  rq_init_comm_if_connected(9, "1")
  rq_init_comm_if_connected(2, "2")
  rq_init_comm_if_connected(3, "3")
  rq_init_comm_if_connected(4, "4")
  rq_print_connected_grippers()
  rq_gripper_communication_thread = run rq_gripper_communication()
  set_closed_norm(100.0, 1)
  set_open_norm(0.0, 1)
  set_closed_mm(0.0, 1)
  set_open_mm(50.0, 1)
  set_closed_norm(100.0, 2)
  set_open_norm(0.0, 2)
  set_closed_mm(0.0, 2)
  set_open_mm(50.0, 2)
  set_closed_norm(100.0, 3)
  set_open_norm(0.0, 3)
  set_closed_mm(0.0, 3)
  set_open_mm(50.0, 3)
  set_closed_norm(100.0, 4)
  set_open_norm(0.0, 4)
  set_closed_mm(0.0, 4)
  set_open_mm(50.0, 4)
  rq_current_limit_enabled = False
  while(not rq_gripper_communication_thread_started):
      sync()
  end
  # end: URCap Installation Node
  global above_grasp_p=p[.151463749910, -.541696949409, .141178566477, .094219767354, -3.102377918313, .016173668201]
  global above_grasp_q=[1.624824047088623, -1.3476700347713013, 1.8017376104937952, -2.0338274441161097, -1.6027372519122522, -0.006902043019429982]
  global at_grasp_p=p[.151456411412, -.541710629189, .044648947210, .094167232389, -3.102376981951, .016262088702]
  global at_grasp_q=[1.6243553161621094, -1.2180383664420624, 1.9187524954425257, -2.2804933987059535, -1.602955166493551, -0.005798641835347951]
  global pass_tray_p=p[.187718005299, -.355766153921, .148265895581, .117471955495, 3.117749481440, -.023888752934]
  global pass_tray_q=[1.7095113166645581, -1.7618856692064426, 2.206533600159921, -2.0337168830746393, -1.5472590068452252, 0.21330219828779456]
  global above_p=p[.200550004174, -.207269798770, .086012234021, .027999624149, 3.115369464841, .006646604504]
  global above_q=[1.8371198687663028, -2.0331563066684026, 2.5463285459008316, -2.0863644147328895, -1.54046586247608, 0.28339987468784766]
  global pick_1_p=p[.200550685402, -.207243112680, .026685871632, 1.785856812100, 2.561238805350, .028538043765]
  global pick_1_q=[1.8360180854797363, -1.8688584766783656, 2.655721966420308, -2.3600183926024383, -1.54055101076235, 1.483529864195182]
  global turn_left_from_p=p[.217155094231, -.247662289880, .015636673097, 1.248001432558, 2.855082939068, -.009943368750]
  global turn_left_to_p=p[.217136235221, -.247633035625, .015613723775, -1.142895665097, 2.911521963648, -.035360810164]
  global very_inclined_p=p[.204088909533, -.207341790181, .029992297833, -1.838165478052, 1.274308683702, -.681817817157]
  global very_inclined_q=[1.0818614959716797, -1.6023737392821253, 2.633673969899313, -1.748885294000143, -0.9851577917682093, -2.6904028097735804]
  global Waypoint_1_p=p[.204646271912, -.207137027515, .060413389860, -2.209248387049, 1.529824787442, -.399222033526]
  global Waypoint_1_q=[1.3692492246627808, -2.017897745172018, 2.631533924733297, -1.8866716823973597, -1.1386383215533655, -2.198780361806051]
  global Waypoint_2_p=p[.204646633947, -.207117303607, .060400735705, 2.031218492370, -1.402721756420, -.557697104030]
  global Waypoint_2_q=[2.4378292560577393, -1.5117061671665688, 2.3492255846606653, -1.9799334011473597, -2.2040918509112757, -0.9229310194598597]
  global Waypoint_3_p=p[.204641926176, -.207147283364, .027003184954, 2.031111530302, -1.402789354928, -.557632875275]
  global Waypoint_3_q=[2.4374465942382812, -1.4238687616637726, 2.3823300043689173, -2.100626131097311, -2.2041776815997522, -0.9223917166339319]
  global Waypoint_5_p=p[.200940609012, -.208521220057, .028794849704, -1.710014056562, 1.186010244159, -.760219738399]
  global Waypoint_5_q=[1.0235025882720947, -1.4368095409921189, 2.5937896410571497, -1.6761061153807582, -0.9735248724566858, -2.82913047472109]
  global Waypoint_6_p=p[.216053995117, -.236413687149, .098791388557, -1.654970470300, 2.048239698933, -.193999891199]
  global Waypoint_6_q=[1.438098430633545, -1.9584604702391566, 2.492446247731344, -1.819071432153219, -1.1232946554767054, -1.558817211781637]
  global incline_from_p=p[.218308125115, -.500893421756, .048170685769, -2.184153264032, 2.228008377241, -.024098614325]
  global incline_to_p=p[.222437586289, -.500865238335, .043608075173, -1.909726804318, 1.946093788457, -.500013830918]
  global Waypoint_4_p=p[.077345856186, -.526444503840, .254497359199, 2.113757942021, -1.933841926219, -.270636769287]
  global Waypoint_4_q=[1.625051498413086, -1.4912703794291993, 1.7121966520892542, -1.844717641870016, -1.8845232168780726, -1.615164581929342]
  global beforehole_p=p[-.066724873844, -.571236623715, .228438737850, 1.497017737305, -1.617613520034, -.828466141634]
  global beforehole_q=[1.6251825971680989, -1.2493833258629223, 1.7962920037571202, -2.0968251742302284, -2.6178372151472837, -1.4260392617096178]
  global athole_p=p[-.093061784839, -.570055041566, .228955616266, 1.497017686755, -1.617613459201, -.828466186119]
  global athole_q=[1.5785684143845495, -1.2561126475132358, 1.8283696329887569, -2.2029137567323094, -2.616872663471543, -1.5189610375905662]
  def calculate_point_to_move_towards(feature, direction, position_distance):
    local posDir=[direction[0], direction[1], direction[2]]
    if (norm(posDir) < 1e-6):
      return get_target_waypoint()
    end
    local direction_vector_normalized=normalize(posDir)
    local displacement_pose=p[direction_vector_normalized[0] * position_distance,direction_vector_normalized[1] * position_distance,direction_vector_normalized[2] * position_distance,0,0,0]
    local wanted_displacement_in_base_frame=pose_sub(pose_trans(feature, displacement_pose), feature)
    return pose_add(get_target_waypoint(), wanted_displacement_in_base_frame)
  end
  global rightturn_from_p=p[-.093068883057, -.570049001092, .228937425705, 1.497031300962, -1.617622590018, -.828512287541]
  global rightturn_to_p=p[-.093055902900, -.570053680269, .228975162208, 1.185666732633, -1.667098189629, -.435688317189]
  global leftturn_from_p=p[-.093048079746, -.570049450859, .228933582576, 1.185754338676, -1.667122132083, -.435696419446]
  global leftturn_to_p=p[-.093068946589, -.570046712102, .228952107442, 1.497042783199, -1.617615149512, -.828519898875]
  global regrasp_point_from_p=p[-.104624192884, -.570099513856, .229070900007, 1.496748297500, -1.617659806479, -.828424735502]
  global regrasp_point_to_p=p[-.090708254877, -.570103474375, .229070367027, 1.496716121525, -1.617687713773, -.828419452272]
  global a_bit_back_p=p[-.059373795033, -.570101759854, .229084958725, 1.496734487750, -1.617649273733, -.828417949027]
  global a_bit_back_q=[1.63824530079538, -1.2506674016840327, 1.7895504324611764, -2.0661997643160825, -2.617569830219447, -1.399815308413035]
  $ 1 "Robot Program"
  $ 2 "MoveJ"
  # begin: URCap Program Node
  #   Source: Robotiq_Grippers, 1.8.1.2444, Robotiq Inc.
  #   Type: Gripper
  $ 3 "Gripper Open (1)"
  if not(gripper_connected[0]):
    popup("Gripper 1 must be connected to run this program.", "No connection", False, True, True)
  end
  if not(rq_is_gripper_activated("1")):
    popup("Gripper 1 is not activated. Go to Installation tab > Gripper to activate it and run the program again.", "Not activated", False, True, True)
  end
  rq_set_pos_spd_for(0, 255, 0, "1")
  rq_wait_pos_spe_for_request(0, 255, 0, "1")
  rq_go_to("1")
  rq_wait("1")
  # end: URCap Program Node
  $ 4 "above_grasp" "breakAfter"
  movej(get_inverse_kin(above_grasp_p, qnear=above_grasp_q), a=1.3962634015954636, v=1.0471975511965976)
  $ 5 "at_grasp" "breakAfter"
  movej(get_inverse_kin(at_grasp_p, qnear=at_grasp_q), a=1.3962634015954636, v=1.0471975511965976)
  # begin: URCap Program Node
  #   Source: Robotiq_Grippers, 1.8.1.2444, Robotiq Inc.
  #   Type: Gripper
  $ 6 "Gripper Close (1)"
  if not(gripper_connected[0]):
    popup("Gripper 1 must be connected to run this program.", "No connection", False, True, True)
  end
  if not(rq_is_gripper_activated("1")):
    popup("Gripper 1 is not activated. Go to Installation tab > Gripper to activate it and run the program again.", "Not activated", False, True, True)
  end
  rq_set_pos_spd_for(255, 255, 255, "1")
  rq_wait_pos_spe_for_request(255, 255, 255, "1")
  rq_go_to("1")
  rq_wait("1")
  # end: URCap Program Node
  $ 7 "Center grasp and turn over"
  $ 8 "MoveL"
  $ 9 "pass_tray" "breakAfter"
  movel(pass_tray_p, a=1.2, v=0.6)
  $ 10 "above" "breakAfter"
  movel(above_p, a=1.2, v=0.6, r=0.05)
  $ 11 "pick_1" "breakAfter"
  movel(pick_1_p, a=1.2, v=0.6)
  # begin: URCap Program Node
  #   Source: Robotiq_Grippers, 1.8.1.2444, Robotiq Inc.
  #   Type: Gripper
  $ 12 "Gripper Move15% (1)"
  if not(gripper_connected[0]):
    popup("Gripper 1 must be connected to run this program.", "No connection", False, True, True)
  end
  if not(rq_is_gripper_activated("1")):
    popup("Gripper 1 is not activated. Go to Installation tab > Gripper to activate it and run the program again.", "Not activated", False, True, True)
  end
  rq_set_pos_spd_for(38, 0, 0, "1")
  rq_wait_pos_spe_for_request(38, 0, 0, "1")
  rq_go_to("1")
  rq_wait("1")
  # end: URCap Program Node
  $ 13 "MoveL"
  $ 14 "turn_left" "breakAfter"
  movel(pose_add(get_target_tcp_pose(), pose_sub(turn_left_to_p, turn_left_from_p)), a=1.2, v=0.6)
  # begin: URCap Program Node
  #   Source: Robotiq_Grippers, 1.8.1.2444, Robotiq Inc.
  #   Type: Gripper
  $ 15 "Gripper Close (1)"
  if not(gripper_connected[0]):
    popup("Gripper 1 must be connected to run this program.", "No connection", False, True, True)
  end
  if not(rq_is_gripper_activated("1")):
    popup("Gripper 1 is not activated. Go to Installation tab > Gripper to activate it and run the program again.", "Not activated", False, True, True)
  end
  rq_set_pos_spd_for(255, 0, 0, "1")
  rq_wait_pos_spe_for_request(255, 0, 0, "1")
  rq_go_to("1")
  rq_wait("1")
  # end: URCap Program Node
  # begin: URCap Program Node
  #   Source: Robotiq_Grippers, 1.8.1.2444, Robotiq Inc.
  #   Type: Gripper
  $ 16 "Gripper Move16% (1)"
  if not(gripper_connected[0]):
    popup("Gripper 1 must be connected to run this program.", "No connection", False, True, True)
  end
  if not(rq_is_gripper_activated("1")):
    popup("Gripper 1 is not activated. Go to Installation tab > Gripper to activate it and run the program again.", "Not activated", False, True, True)
  end
  rq_set_pos_spd_for(42, 255, 255, "1")
  rq_wait_pos_spe_for_request(42, 255, 255, "1")
  rq_go_to("1")
  rq_wait("1")
  # end: URCap Program Node
  $ 17 "MoveL"
  $ 18 "turn_left" "breakAfter"
  movel(pose_add(get_target_tcp_pose(), pose_sub(turn_left_to_p, turn_left_from_p)), a=1.2, v=0.6)
  $ 20 "very_inclined" "breakAfter"
  movel(very_inclined_p, a=1.2, v=0.6)
  # begin: URCap Program Node
  #   Source: Robotiq_Grippers, 1.8.1.2444, Robotiq Inc.
  #   Type: Gripper
  $ 21 "Gripper Close (1)"
  if not(gripper_connected[0]):
    popup("Gripper 1 must be connected to run this program.", "No connection", False, True, True)
  end
  if not(rq_is_gripper_activated("1")):
    popup("Gripper 1 is not activated. Go to Installation tab > Gripper to activate it and run the program again.", "Not activated", False, True, True)
  end
  rq_set_pos_spd_for(255, 255, 255, "1")
  rq_wait_pos_spe_for_request(255, 255, 255, "1")
  rq_go_to("1")
  rq_wait("1")
  # end: URCap Program Node
  $ 22 "Turn over"
  $ 23 "MoveL"
  $ 24 "Waypoint_1" "breakAfter"
  movel(Waypoint_1_p, a=1.2, v=0.25)
  $ 25 "Waypoint_2" "breakAfter"
  movel(Waypoint_2_p, a=1.2, v=0.25)
  $ 26 "Waypoint_3" "breakAfter"
  movel(Waypoint_3_p, a=1.2, v=0.25)
  # begin: URCap Program Node
  #   Source: Robotiq_Grippers, 1.8.1.2444, Robotiq Inc.
  #   Type: Gripper
  $ 27 "Gripper Move16% (1)"
  if not(gripper_connected[0]):
    popup("Gripper 1 must be connected to run this program.", "No connection", False, True, True)
  end
  if not(rq_is_gripper_activated("1")):
    popup("Gripper 1 is not activated. Go to Installation tab > Gripper to activate it and run the program again.", "Not activated", False, True, True)
  end
  rq_set_pos_spd_for(42, 255, 255, "1")
  rq_wait_pos_spe_for_request(42, 255, 255, "1")
  rq_go_to("1")
  rq_wait("1")
  # end: URCap Program Node
  $ 28 "Waypoint_5" "breakAfter"
  movel(Waypoint_5_p, a=1.2, v=0.25)
  # begin: URCap Program Node
  #   Source: Robotiq_Grippers, 1.8.1.2444, Robotiq Inc.
  #   Type: Gripper
  $ 29 "Gripper Close (1)"
  if not(gripper_connected[0]):
    popup("Gripper 1 must be connected to run this program.", "No connection", False, True, True)
  end
  if not(rq_is_gripper_activated("1")):
    popup("Gripper 1 is not activated. Go to Installation tab > Gripper to activate it and run the program again.", "Not activated", False, True, True)
  end
  rq_set_pos_spd_for(255, 255, 255, "1")
  rq_wait_pos_spe_for_request(255, 255, 255, "1")
  rq_go_to("1")
  rq_wait("1")
  # end: URCap Program Node
  $ 30 "Waypoint_6" "breakAfter"
  movel(Waypoint_6_p, a=1.2, v=0.25)
  $ 31 "Center grasp and pick inclined"
  $ 32 "MoveL"
  $ 34 "above" "breakAfter"
  movel(above_p, a=1.2, v=0.6, r=0.034)
  $ 35 "pick_1" "breakAfter"
  movel(pick_1_p, a=1.2, v=0.6)
  # begin: URCap Program Node
  #   Source: Robotiq_Grippers, 1.8.1.2444, Robotiq Inc.
  #   Type: Gripper
  $ 36 "Gripper Move15% (1)"
  if not(gripper_connected[0]):
    popup("Gripper 1 must be connected to run this program.", "No connection", False, True, True)
  end
  if not(rq_is_gripper_activated("1")):
    popup("Gripper 1 is not activated. Go to Installation tab > Gripper to activate it and run the program again.", "Not activated", False, True, True)
  end
  rq_set_pos_spd_for(38, 0, 0, "1")
  rq_wait_pos_spe_for_request(38, 0, 0, "1")
  rq_go_to("1")
  rq_wait("1")
  # end: URCap Program Node
  $ 37 "MoveL"
  $ 38 "turn_left" "breakAfter"
  movel(pose_add(get_target_tcp_pose(), pose_sub(turn_left_to_p, turn_left_from_p)), a=1.2, v=0.6)
  # begin: URCap Program Node
  #   Source: Robotiq_Grippers, 1.8.1.2444, Robotiq Inc.
  #   Type: Gripper
  $ 40 "Gripper Close (1)"
  if not(gripper_connected[0]):
    popup("Gripper 1 must be connected to run this program.", "No connection", False, True, True)
  end
  if not(rq_is_gripper_activated("1")):
    popup("Gripper 1 is not activated. Go to Installation tab > Gripper to activate it and run the program again.", "Not activated", False, True, True)
  end
  rq_set_pos_spd_for(255, 0, 0, "1")
  rq_wait_pos_spe_for_request(255, 0, 0, "1")
  rq_go_to("1")
  rq_wait("1")
  # end: URCap Program Node
  # begin: URCap Program Node
  #   Source: Robotiq_Grippers, 1.8.1.2444, Robotiq Inc.
  #   Type: Gripper
  $ 41 "Gripper Move16% (1)"
  if not(gripper_connected[0]):
    popup("Gripper 1 must be connected to run this program.", "No connection", False, True, True)
  end
  if not(rq_is_gripper_activated("1")):
    popup("Gripper 1 is not activated. Go to Installation tab > Gripper to activate it and run the program again.", "Not activated", False, True, True)
  end
  rq_set_pos_spd_for(42, 255, 255, "1")
  rq_wait_pos_spe_for_request(42, 255, 255, "1")
  rq_go_to("1")
  rq_wait("1")
  # end: URCap Program Node
  $ 42 "MoveL"
  $ 44 "turn_left" "breakAfter"
  movel(pose_add(get_target_tcp_pose(), pose_sub(turn_left_to_p, turn_left_from_p)), a=1.2, v=0.6)
  $ 45 "incline" "breakAfter"
  movel(pose_add(get_target_tcp_pose(), pose_sub(incline_to_p, incline_from_p)), a=1.2, v=0.6)
  # begin: URCap Program Node
  #   Source: Robotiq_Grippers, 1.8.1.2444, Robotiq Inc.
  #   Type: Gripper
  $ 46 "Gripper Close (1)"
  if not(gripper_connected[0]):
    popup("Gripper 1 must be connected to run this program.", "No connection", False, True, True)
  end
  if not(rq_is_gripper_activated("1")):
    popup("Gripper 1 is not activated. Go to Installation tab > Gripper to activate it and run the program again.", "Not activated", False, True, True)
  end
  rq_set_pos_spd_for(255, 255, 255, "1")
  rq_wait_pos_spe_for_request(255, 255, 255, "1")
  rq_go_to("1")
  rq_wait("1")
  # end: URCap Program Node
  $ 47 "MoveL"
  $ 48 "above" "breakAfter"
  set_tcp(p[0.0,0.0,0.165,0.0,0.0,0.0])
  movel(above_p, a=1.2, v=0.6)
  $ 49 "MoveJ"
  $ 50 "Waypoint_4" "breakAfter"
  set_tcp(p[0.0,0.0,0.165,0.0,0.0,0.0])
  movej(get_inverse_kin(Waypoint_4_p, qnear=Waypoint_4_q), a=6.283185307179586, v=3.141592653589793, r=0.05)
  $ 51 "beforehole" "breakAfter"
  set_tcp(p[0.0,0.0,0.165,0.0,0.0,0.0])
  movej(get_inverse_kin(beforehole_p, qnear=beforehole_q), a=6.283185307179586, v=3.141592653589793)
  $ 52 "athole" "breakAfter"
  set_tcp(p[0.0,0.0,0.165,0.0,0.0,0.0])
  movej(get_inverse_kin(athole_p, qnear=athole_q), a=6.283185307179586, v=3.141592653589793)
  $ 53 "first insert"
  $ 54 "loop_1≔0"
  global loop_1=0
  $ 55 "tcp_p≔get_actual_tcp_pose()"
  global tcp_p= get_actual_tcp_pose ()
  $ 56 "Force"
  sleep(0.02)
  zero_ftsensor()
  force_mode(p[0.0,0.0,0.0,0.0,0.0,0.0], [1, 0, 0, 0, 0, 0], [-5.0, 0.0, 10.0, 0.0, 0.0, 0.0], 2, [0.01, 0.1, 0.1, 0.3490658503988659, 0.3490658503988659, 0.3490658503988659])
  $ 57 "Loop ( tcp_p[0] > -0.095) and  (loop_1 < 1) " "noBreak"
  while (( tcp_p[0] > -0.095)  and   (loop_1 < 1) ):
    $ 58 "MoveL" "noBreak"
    $ 59 "Direction: Base Y+" "noBreak"
    global move_thread_flag_59=0
    thread move_thread_59():
      enter_critical
      move_thread_flag_59 = 1
      local towardsPos=calculate_point_to_move_towards(p[0.0,0.0,0.0,0.0,0.0,0.0], [0.0,1.0,0.0], 0.001)
      movel(towardsPos, a=0.02, v=0.005)
      move_thread_flag_59 = 2
      exit_critical
    end
    move_thread_flag_59 = 0
    move_thread_han_59 = run move_thread_59()
    while (True):
      sleep(1.0E-10)
      if (move_thread_flag_59 > 1):
        join move_thread_han_59
        $ 60 "Until (distance)" "noBreak"
        break
      end
      sync()
    end
    $ 61 "Direction: Base Z-" "noBreak"
    global move_thread_flag_61=0
    thread move_thread_61():
      enter_critical
      move_thread_flag_61 = 1
      local towardsPos=calculate_point_to_move_towards(p[0.0,0.0,0.0,0.0,0.0,0.0], [0.0,0.0,-1.0], 0.001)
      movel(towardsPos, a=0.02, v=0.005)
      move_thread_flag_61 = 2
      exit_critical
    end
    move_thread_flag_61 = 0
    move_thread_han_61 = run move_thread_61()
    while (True):
      sleep(1.0E-10)
      if (move_thread_flag_61 > 1):
        join move_thread_han_61
        $ 62 "Until (distance)" "noBreak"
        break
      end
      sync()
    end
    $ 63 "tcp_p≔get_actual_tcp_pose()" "noBreak"
    global tcp_p= get_actual_tcp_pose ()
    $ 64 "Direction: Base Y-" "noBreak"
    global move_thread_flag_64=0
    thread move_thread_64():
      enter_critical
      move_thread_flag_64 = 1
      local towardsPos=calculate_point_to_move_towards(p[0.0,0.0,0.0,0.0,0.0,0.0], [0.0,-1.0,0.0], 0.001)
      movel(towardsPos, a=0.02, v=0.005)
      move_thread_flag_64 = 2
      exit_critical
    end
    move_thread_flag_64 = 0
    move_thread_han_64 = run move_thread_64()
    while (True):
      sleep(1.0E-10)
      if (move_thread_flag_64 > 1):
        join move_thread_han_64
        $ 65 "Until (distance)" "noBreak"
        break
      end
      sync()
    end
    $ 66 "Direction: Base Y-" "noBreak"
    global move_thread_flag_66=0
    thread move_thread_66():
      enter_critical
      move_thread_flag_66 = 1
      local towardsPos=calculate_point_to_move_towards(p[0.0,0.0,0.0,0.0,0.0,0.0], [0.0,-1.0,0.0], 0.001)
      movel(towardsPos, a=0.02, v=0.005)
      move_thread_flag_66 = 2
      exit_critical
    end
    move_thread_flag_66 = 0
    move_thread_han_66 = run move_thread_66()
    while (True):
      sleep(1.0E-10)
      if (move_thread_flag_66 > 1):
        join move_thread_han_66
        $ 67 "Until (distance)" "noBreak"
        break
      end
      sync()
    end
    $ 68 "tcp_p≔get_actual_tcp_pose()" "noBreak"
    global tcp_p= get_actual_tcp_pose ()
    $ 69 "Direction: Base Z+" "noBreak"
    global move_thread_flag_69=0
    thread move_thread_69():
      enter_critical
      move_thread_flag_69 = 1
      local towardsPos=calculate_point_to_move_towards(p[0.0,0.0,0.0,0.0,0.0,0.0], [0.0,0.0,1.0], 0.001)
      movel(towardsPos, a=0.02, v=0.005)
      move_thread_flag_69 = 2
      exit_critical
    end
    move_thread_flag_69 = 0
    move_thread_han_69 = run move_thread_69()
    while (True):
      sleep(1.0E-10)
      if (move_thread_flag_69 > 1):
        join move_thread_han_69
        $ 70 "Until (distance)" "noBreak"
        break
      end
      sync()
    end
    $ 71 "Direction: Base Y+" "noBreak"
    global move_thread_flag_71=0
    thread move_thread_71():
      enter_critical
      move_thread_flag_71 = 1
      local towardsPos=calculate_point_to_move_towards(p[0.0,0.0,0.0,0.0,0.0,0.0], [0.0,1.0,0.0], 0.001)
      movel(towardsPos, a=0.02, v=0.005)
      move_thread_flag_71 = 2
      exit_critical
    end
    move_thread_flag_71 = 0
    move_thread_han_71 = run move_thread_71()
    while (True):
      sleep(1.0E-10)
      if (move_thread_flag_71 > 1):
        join move_thread_han_71
        $ 72 "Until (distance)" "noBreak"
        break
      end
      sync()
    end
    $ 73 "tcp_p≔get_actual_tcp_pose()" "noBreak"
    global tcp_p= get_actual_tcp_pose ()
    $ 74 "Direction: Base Y+" "noBreak"
    global move_thread_flag_74=0
    thread move_thread_74():
      enter_critical
      move_thread_flag_74 = 1
      local towardsPos=calculate_point_to_move_towards(p[0.0,0.0,0.0,0.0,0.0,0.0], [0.0,1.0,0.0], 0.001)
      movel(towardsPos, a=0.02, v=0.005)
      move_thread_flag_74 = 2
      exit_critical
    end
    move_thread_flag_74 = 0
    move_thread_han_74 = run move_thread_74()
    while (True):
      sleep(1.0E-10)
      if (move_thread_flag_74 > 1):
        join move_thread_han_74
        $ 75 "Until (distance)" "noBreak"
        break
      end
      sync()
    end
    $ 76 "Direction: Base Z+" "noBreak"
    global move_thread_flag_76=0
    thread move_thread_76():
      enter_critical
      move_thread_flag_76 = 1
      local towardsPos=calculate_point_to_move_towards(p[0.0,0.0,0.0,0.0,0.0,0.0], [0.0,0.0,1.0], 0.001)
      movel(towardsPos, a=0.02, v=0.005)
      move_thread_flag_76 = 2
      exit_critical
    end
    move_thread_flag_76 = 0
    move_thread_han_76 = run move_thread_76()
    while (True):
      sleep(1.0E-10)
      if (move_thread_flag_76 > 1):
        join move_thread_han_76
        $ 77 "Until (distance)" "noBreak"
        break
      end
      sync()
    end
    $ 78 "tcp_p≔get_actual_tcp_pose()" "noBreak"
    global tcp_p= get_actual_tcp_pose ()
    $ 79 "Direction: Base Y-" "noBreak"
    global move_thread_flag_79=0
    thread move_thread_79():
      enter_critical
      move_thread_flag_79 = 1
      local towardsPos=calculate_point_to_move_towards(p[0.0,0.0,0.0,0.0,0.0,0.0], [0.0,-1.0,0.0], 0.001)
      movel(towardsPos, a=0.02, v=0.005)
      move_thread_flag_79 = 2
      exit_critical
    end
    move_thread_flag_79 = 0
    move_thread_han_79 = run move_thread_79()
    while (True):
      sleep(1.0E-10)
      if (move_thread_flag_79 > 1):
        join move_thread_han_79
        $ 80 "Until (distance)" "noBreak"
        break
      end
      sync()
    end
    $ 81 "Direction: Base Y-" "noBreak"
    global move_thread_flag_81=0
    thread move_thread_81():
      enter_critical
      move_thread_flag_81 = 1
      local towardsPos=calculate_point_to_move_towards(p[0.0,0.0,0.0,0.0,0.0,0.0], [0.0,-1.0,0.0], 0.001)
      movel(towardsPos, a=0.02, v=0.005)
      move_thread_flag_81 = 2
      exit_critical
    end
    move_thread_flag_81 = 0
    move_thread_han_81 = run move_thread_81()
    while (True):
      sleep(1.0E-10)
      if (move_thread_flag_81 > 1):
        join move_thread_han_81
        $ 82 "Until (distance)" "noBreak"
        break
      end
      sync()
    end
    $ 83 "tcp_p≔get_actual_tcp_pose()" "noBreak"
    global tcp_p= get_actual_tcp_pose ()
    $ 84 "Direction: Base Z-" "noBreak"
    global move_thread_flag_84=0
    thread move_thread_84():
      enter_critical
      move_thread_flag_84 = 1
      local towardsPos=calculate_point_to_move_towards(p[0.0,0.0,0.0,0.0,0.0,0.0], [0.0,0.0,-1.0], 0.001)
      movel(towardsPos, a=0.02, v=0.005)
      move_thread_flag_84 = 2
      exit_critical
    end
    move_thread_flag_84 = 0
    move_thread_han_84 = run move_thread_84()
    while (True):
      sleep(1.0E-10)
      if (move_thread_flag_84 > 1):
        join move_thread_han_84
        $ 85 "Until (distance)" "noBreak"
        break
      end
      sync()
    end
    $ 86 "Direction: Base Y+" "noBreak"
    global move_thread_flag_86=0
    thread move_thread_86():
      enter_critical
      move_thread_flag_86 = 1
      local towardsPos=calculate_point_to_move_towards(p[0.0,0.0,0.0,0.0,0.0,0.0], [0.0,1.0,0.0], 0.001)
      movel(towardsPos, a=0.02, v=0.005)
      move_thread_flag_86 = 2
      exit_critical
    end
    move_thread_flag_86 = 0
    move_thread_han_86 = run move_thread_86()
    while (True):
      sleep(1.0E-10)
      if (move_thread_flag_86 > 1):
        join move_thread_han_86
        $ 87 "Until (distance)" "noBreak"
        break
      end
      sync()
    end
    $ 88 "tcp_p≔get_actual_tcp_pose()" "noBreak"
    global tcp_p= get_actual_tcp_pose ()
    $ 89 "MoveL" "noBreak"
    $ 90 "rightturn" "noBreak"
    set_tcp(p[0.0,0.0,0.165,0.0,0.0,0.0])
    movel(pose_add(get_target_tcp_pose(), pose_sub(rightturn_to_p, rightturn_from_p)), a=0.2, v=0.05)
    $ 91 "tcp_p≔get_actual_tcp_pose()" "noBreak"
    global tcp_p= get_actual_tcp_pose ()
    $ 92 "leftturn" "noBreak"
    set_tcp(p[0.0,0.0,0.165,0.0,0.0,0.0])
    movel(pose_add(get_target_tcp_pose(), pose_sub(leftturn_to_p, leftturn_from_p)), a=0.2, v=0.05)
    $ 93 "tcp_p≔get_actual_tcp_pose()" "noBreak"
    global tcp_p= get_actual_tcp_pose ()
    $ 94 "leftturn" "noBreak"
    set_tcp(p[0.0,0.0,0.165,0.0,0.0,0.0])
    movel(pose_add(get_target_tcp_pose(), pose_sub(leftturn_to_p, leftturn_from_p)), a=0.2, v=0.05)
    $ 95 "tcp_p≔get_actual_tcp_pose()" "noBreak"
    global tcp_p= get_actual_tcp_pose ()
    $ 96 "rightturn" "noBreak"
    set_tcp(p[0.0,0.0,0.165,0.0,0.0,0.0])
    movel(pose_add(get_target_tcp_pose(), pose_sub(rightturn_to_p, rightturn_from_p)), a=0.2, v=0.05)
    $ 97 "tcp_p≔get_actual_tcp_pose()" "noBreak"
    global tcp_p= get_actual_tcp_pose ()
    $ 98 "loop_1≔loop_1+1" "noBreak"
    global loop_1=loop_1+1
    $ 99 "tcp_p≔get_actual_tcp_pose()" "noBreak"
    global tcp_p= get_actual_tcp_pose ()
  end
  end_force_mode()
  stopl(5.0)
  # begin: URCap Program Node
  #   Source: Robotiq_Grippers, 1.8.1.2444, Robotiq Inc.
  #   Type: Gripper
  $ 100 "Gripper Open (1)"
  if not(gripper_connected[0]):
    popup("Gripper 1 must be connected to run this program.", "No connection", False, True, True)
  end
  if not(rq_is_gripper_activated("1")):
    popup("Gripper 1 is not activated. Go to Installation tab > Gripper to activate it and run the program again.", "Not activated", False, True, True)
  end
  rq_set_pos_spd_for(0, 255, 0, "1")
  rq_wait_pos_spe_for_request(0, 255, 0, "1")
  rq_go_to("1")
  rq_wait("1")
  # end: URCap Program Node
  $ 101 "MoveJ"
  $ 102 "regrasp_point" "breakAfter"
  set_tcp(p[0.0,0.0,0.165,0.0,0.0,0.0])
  movej(pose_add(get_target_tcp_pose(), pose_sub(regrasp_point_to_p, regrasp_point_from_p)), a=1.3962634015954636, v=1.0471975511965976)
  # begin: URCap Program Node
  #   Source: Robotiq_Grippers, 1.8.1.2444, Robotiq Inc.
  #   Type: Gripper
  $ 103 "Gripper Close (1)"
  if not(gripper_connected[0]):
    popup("Gripper 1 must be connected to run this program.", "No connection", False, True, True)
  end
  if not(rq_is_gripper_activated("1")):
    popup("Gripper 1 is not activated. Go to Installation tab > Gripper to activate it and run the program again.", "Not activated", False, True, True)
  end
  rq_set_pos_spd_for(255, 255, 255, "1")
  rq_wait_pos_spe_for_request(255, 255, 255, "1")
  rq_go_to("1")
  rq_wait("1")
  # end: URCap Program Node
  $ 104 "If rq_current_pos_mm()<10"
  if ( rq_current_pos_mm ()<10):
    $ 105 "'Gripper fully closed = bearing not inserted!! Stopping.'"
    # 'Gripper fully closed = bearing not inserted!! Stopping.'
    $ 106 "MoveL"
    $ 107 "Direction: Base X+"
    global move_thread_flag_107=0
    thread move_thread_107():
      enter_critical
      move_thread_flag_107 = 1
      local towardsPos=calculate_point_to_move_towards(p[0.0,0.0,0.0,0.0,0.0,0.0], [1.0,0.0,0.0], 0.1)
      movel(towardsPos, a=0.06, v=0.1)
      move_thread_flag_107 = 2
      exit_critical
    end
    move_thread_flag_107 = 0
    move_thread_han_107 = run move_thread_107()
    while (True):
      sleep(1.0E-10)
      if (move_thread_flag_107 > 1):
        join move_thread_han_107
        $ 108 "Until (distance)"
        break
      end
      sync()
    end
    $ 109 "Halt"
    halt
  end
  $ 110 "second insert"
  $ 111 "loop_1≔0"
  global loop_1=0
  $ 112 "tcp_p≔get_actual_tcp_pose()"
  global tcp_p= get_actual_tcp_pose ()
  $ 113 "Force"
  sleep(0.02)
  zero_ftsensor()
  force_mode(p[0.0,0.0,0.0,0.0,0.0,0.0], [1, 0, 0, 0, 0, 0], [-5.0, 0.0, 10.0, 0.0, 0.0, 0.0], 2, [0.01, 0.1, 0.1, 0.3490658503988659, 0.3490658503988659, 0.3490658503988659])
  $ 114 "Loop ( tcp_p[0] > -0.095) and  (loop_1 < 1) " "noBreak"
  while (( tcp_p[0] > -0.095)  and   (loop_1 < 1) ):
    $ 115 "MoveL" "noBreak"
    $ 116 "rightturn" "noBreak"
    set_tcp(p[0.0,0.0,0.165,0.0,0.0,0.0])
    movel(pose_add(get_target_tcp_pose(), pose_sub(rightturn_to_p, rightturn_from_p)), a=0.2, v=0.05)
    $ 117 "tcp_p≔get_actual_tcp_pose()" "noBreak"
    global tcp_p= get_actual_tcp_pose ()
    $ 118 "leftturn" "noBreak"
    set_tcp(p[0.0,0.0,0.165,0.0,0.0,0.0])
    movel(pose_add(get_target_tcp_pose(), pose_sub(leftturn_to_p, leftturn_from_p)), a=0.2, v=0.05)
    $ 119 "tcp_p≔get_actual_tcp_pose()" "noBreak"
    global tcp_p= get_actual_tcp_pose ()
    $ 120 "leftturn" "noBreak"
    set_tcp(p[0.0,0.0,0.165,0.0,0.0,0.0])
    movel(pose_add(get_target_tcp_pose(), pose_sub(leftturn_to_p, leftturn_from_p)), a=0.2, v=0.05)
    $ 121 "tcp_p≔get_actual_tcp_pose()" "noBreak"
    global tcp_p= get_actual_tcp_pose ()
    $ 122 "rightturn" "noBreak"
    set_tcp(p[0.0,0.0,0.165,0.0,0.0,0.0])
    movel(pose_add(get_target_tcp_pose(), pose_sub(rightturn_to_p, rightturn_from_p)), a=0.2, v=0.05)
    $ 123 "tcp_p≔get_actual_tcp_pose()" "noBreak"
    global tcp_p= get_actual_tcp_pose ()
    $ 124 "loop_1≔loop_1+1" "noBreak"
    global loop_1=loop_1+1
    $ 125 "tcp_p≔get_actual_tcp_pose()" "noBreak"
    global tcp_p= get_actual_tcp_pose ()
  end
  end_force_mode()
  stopl(5.0)
  # begin: URCap Program Node
  #   Source: Robotiq_Grippers, 1.8.1.2444, Robotiq Inc.
  #   Type: Gripper
  $ 126 "Gripper Open (1)"
  if not(gripper_connected[0]):
    popup("Gripper 1 must be connected to run this program.", "No connection", False, True, True)
  end
  if not(rq_is_gripper_activated("1")):
    popup("Gripper 1 is not activated. Go to Installation tab > Gripper to activate it and run the program again.", "Not activated", False, True, True)
  end
  rq_set_pos_spd_for(0, 255, 0, "1")
  rq_wait_pos_spe_for_request(0, 255, 0, "1")
  rq_go_to("1")
  rq_wait("1")
  # end: URCap Program Node
  $ 140 "MoveJ"
  $ 141 "a_bit_back" "breakAfter"
  set_tcp(p[0.0,0.0,0.165,0.0,0.0,0.0])
  movej(get_inverse_kin(a_bit_back_p, qnear=a_bit_back_q), a=1.3962634015954636, v=1.0471975511965976)
  # begin: URCap Program Node
  #   Source: Robotiq_Grippers, 1.8.1.2444, Robotiq Inc.
  #   Type: Gripper
  $ 142 "Gripper Open (1)"
  if not(gripper_connected[0]):
    popup("Gripper 1 must be connected to run this program.", "No connection", False, True, True)
  end
  if not(rq_is_gripper_activated("1")):
    popup("Gripper 1 is not activated. Go to Installation tab > Gripper to activate it and run the program again.", "Not activated", False, True, True)
  end
  rq_set_pos_spd_for(0, 255, 0, "1")
  rq_wait_pos_spe_for_request(0, 255, 0, "1")
  rq_go_to("1")
  rq_wait("1")
  # end: URCap Program Node
end
